(* Schneider Machine Expert - Basic project Comparação de valores IO analógicas, file version 3.0.0.0 *)
(* CompanyInformations: Name=Sidney, PhoneNumber=(27) 99648-9123, Street=Rua dos Tupinambás, City=Belo Horizonte, ZipCode=30120040, State=Minas Gerais, Country=Brasil, WebSite=https://sidney-personal-portfolio.netlify.app *)
(* ProjectInformations: Name=Comparador de valores, Description=Exercício simples de comparação de valores, para fixação do conteúdo didático. *)
(* UserInformations: LastName=Sidney, FirstName=Junior, CellNumber=(27 ) 99648-9123, Email=sidneyteodoroaraujojunior2002@gmail.com, Street=Rua dos Tupinambás, City=Belo Horizonte, ZipCode=30120040, State=Minas Gerais, Country=Brasil *)

HARDWARE
  Cpu 0: TM221CE40R
  EthernetConfiguration: NetworkName=M221, IpAllocationMode=FixedAddress, IpAddress=0.0.0.0, SubnetMask=0.0.0.0
  SerialLineConfiguration: Baud=Baud19200, Parity=ParityEven, DataBits=DataBits8, StopBits=StopBits1, PhysicalMedium=PhysicalMediumRs485, TransmissionMode=TransmissionModeModbusRtu, SlaveId=1, Addressing=SlaveAddressing
  MastTask: UsePeriodScanMode=false, PeriodScan=100
  FastTask: Period=255
  CpuBehavior: StartingMode=StartAsPreviousState, AutoSaveRamOnEeprom=true, WatchdogPeriod=250

SYMBOLS  (address, symbol, comment, settings)
  %IW0.0      [Type=Type_0_10V, Scope=Scope_Normal, Minimum=0, Maximum=1000]
  %IW0.1      [Type=Type_0_10V, Scope=Scope_Normal, Minimum=0, Maximum=1000]

POU Novo POU
  (* SectionNumber=1 *)

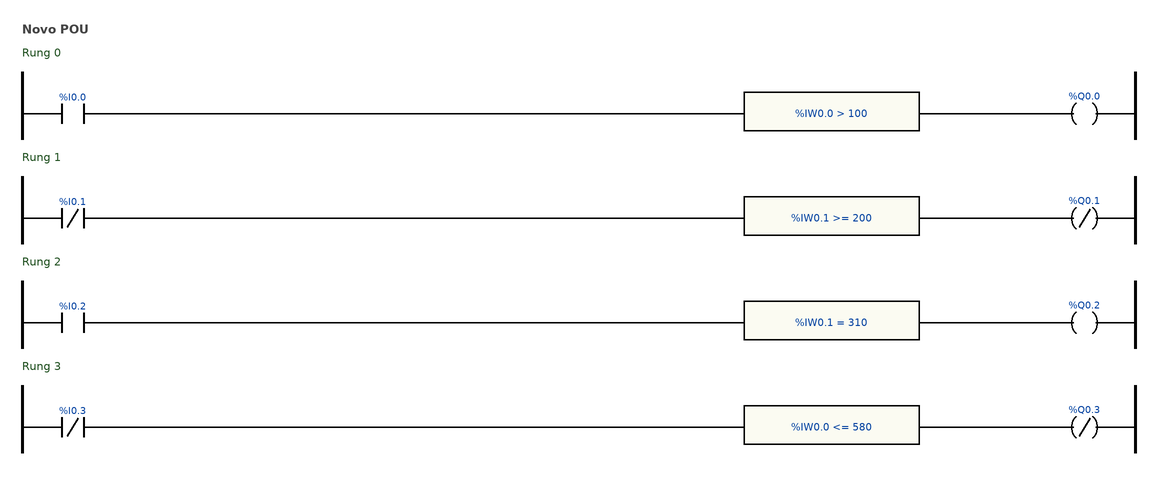

// Rung 0
  LD %I0.0
  AND [ %IW0.0 > 100 ]
  ST %Q0.0
  // as ST:
  //   %Q0.0 := %I0.0 AND %IW0.0 > 100;

// Rung 1
  LDN %I0.1
  AND [ %IW0.1 >= 200 ]
  STN %Q0.1
  // as ST:
  //   %Q0.1 := NOT (NOT %I0.1 AND %IW0.1 >= 200);

// Rung 2
  LD %I0.2
  AND [ %IW0.1 = 310 ]
  ST %Q0.2
  // as ST:
  //   %Q0.2 := %I0.2 AND %IW0.1 = 310;

// Rung 3
  LDN %I0.3
  AND [ %IW0.0 <= 580 ]
  STN %Q0.3
  // as ST:
  //   %Q0.3 := NOT (NOT %I0.3 AND %IW0.0 <= 580);
